// TIA Portal project "2022.05.22_制作模板" (V17)

(* hardware
DEVICE "S7-1500/ET200MP station_1"  S7-1500 station
   slot 0: "导轨_0"  Rack  6ES7 590-1***0-0AA0
   slot 1: "PLC_1500"  CPU 1516-3 PN/DP  6ES7 516-3AN00-0AB0  V1.7
      slot 3: "CPU 显示_1"  6ES7591-1BA00-0AA0
      slot 32768: "PROFINET 接口_1"  X1
         slot 32769: "端口_1"  X1 P1
         slot 32770: "端口_2"  X1 P2
      slot 33024: "PROFINET 接口_2"  X2
         slot 33025: "端口_1"  X2 P1
      slot 33280: "DP 接口_1"  X3
DEVICE "HMI_1"  TP1200 Comfort
   slot 0: "HMI_1"  TP1200 Comfort  6AV2 124-0MC01-0AX0  17.0.0.0
   slot 1: "HMI_RT_1"  TP1200 Comfort  6AV2 124-0MC01-0AX0  17.0.0.0
   slot 5: "HMI_1.IE_CP_1"  PROFINET Interface  17.0.0.0
      slot 1: "PROFINET Interface_1"  PROFINET Interface
         slot 1: "Port_1"  Port
         slot 2: "Port_2"  Port
   slot 7: "HMI_1.MPI/DP_CP_1"  MPI/DP Interface  17.0.0.0
*)

// ===== PLC "PLC_1500"  CPU 1516-3 PN/DP =====

DATA_BLOCK "DATE_AND_TIME"   // DB1
{ S7_Optimized_Access := 'TRUE' }
VERSION : 0.1
   VAR
      "time" : Date_And_Time;
      time_ret : Int;
   END_VAR
BEGIN
END_DATA_BLOCK

ORGANIZATION_BLOCK "Main"   // OB1, LAD, ProgramCycle
TITLE = "Main Program Sweep (Cycle)"
{ S7_Optimized_Access := 'TRUE' }
VERSION : 0.1
   VAR_INPUT
      Initial_Call : Bool;   // Initial call of this OB
      Remanence : Bool;   // =True, if remanent data are available
   END_VAR
BEGIN

REGION Network 1
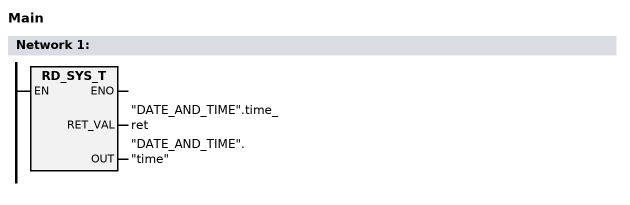
   "DATE_AND_TIME".time_ret := RD_SYS_T(OUT => "DATE_AND_TIME"."time");
END_REGION
END_ORGANIZATION_BLOCK

(* ===== HMI "HMI_RT_1" =====
system functions are stored by id; their names below are inferred from use
connection "PLC_1500": ETHERNET, S7_1500_OMS
connection "Connection_1": ETHERNET, S7_1500_OMS

HMI tags "默认变量表"
   "DATE_AND_TIME_time_ret" : Int = PLC "DATE_AND_TIME".time_ret, 1 s

HMI tags "外部变量"
   "DATE_AND_TIME_time" : Date_And_Time = PLC "DATE_AND_TIME".time, 1 s

HMI tags "内部变量"
   "画面切换颜色" : Int, internal

screen "首页" 1280x740, template "模板_1"
   on GenerateScreen: SetTag("画面切换颜色", 1)

Template "模板_1" 1280x740
   Button "Template_Button_13" at 81,679 size 153x59; TextOff '用户界面1'
      on Release: ActivateScreen("用户界面1", 0); SetTag("画面切换颜色", 2)
      Appearance <- "画面切换颜色"
   Button "退出" at 1200,679 size 78x59; TextOff '退出'; PictureOff "ExitRuntime_TP1200_Comfort_TR"; PictureOn "ExitRuntime_TP1200_Comfort_TR"
      on Release: StopRuntime(0)
   Button "起始画面" at 1,679 size 78x59; TextOff '起始画面'; PictureOff "NavigateHome_TP1200_Comfort_TR"; PictureOn "NavigateHome_TP1200_Comfort_TR"
      on Release: SetTag("画面切换颜色", 1); ActivateScreen("首页", 0)
      Appearance <- "画面切换颜色"
   Button "Template_Button_1" at 236,679 size 153x59; TextOn '用户界面2'; TextOff '用户界面2'
      on Release: ActivateScreen("用户界面2", 0); SetTag("画面切换颜色", 3)
      Appearance <- "画面切换颜色"
   Button "Template_Button_2" at 393,678 size 153x59; TextOn '测试界面'; TextOff '测试界面'
      on Release: ActivateScreen("测试界面", 0); SetTag("画面切换颜色", 4)
      Appearance <- "画面切换颜色"
   Button "Template_Button_3" at 551,678 size 153x59; TextOn '用户管理界面'; TextOff '用户管理界面'
      on Release: ActivateScreen("用户管理界面", 0); SetTag("画面切换颜色", 5)
      Appearance <- "画面切换颜色"
   Button "Template_Button_4" at 710,678 size 153x59; TextOn '报警管理界面'; TextOff '报警管理界面'
      on Release: ActivateScreen("报警视图画面", 0); SetTag("画面切换颜色", 6)
      Appearance <- "画面切换颜色"
   Button "Template_Button_5" at 868,678 size 153x59; TextOn '系统诊断界面'; TextOff '系统诊断界面'
      on Release: ActivateScreen("系统诊断界面", 0); SetTag("画面切换颜色", 7)
      Appearance <- "画面切换颜色"
   Button "Template_Button_6" at 1027,678 size 153x59; TextOn '备用界面'; TextOff '备用界面'
      on Release: ActivateScreen("备用界面", 0); SetTag("画面切换颜色", 8)
      Appearance <- "画面切换颜色"

screen "用户管理界面" 1280x740, template "模板_1"
   UserView "用户视图_1" at 2,2 size 1277x676

screen "报警视图画面" 1280x740, template "模板_1"
   AlarmView "报警视图_1" at 0,0 size 1280x676

screen "系统诊断界面" 1280x740, template "模板_1"
   SysDiagControl "系统诊断视图_1" at 0,2 size 1278x676
*)